    PROC rMoveWeld()
        IF nMode=1 THEN
            stCommand:="Weld1";
            WaitUntil stReact=["WeldOk","WeldOk","WeldOk"]OR stReact=["Error_Arc_Touch","Error_Arc_Touch","Error_Arc_Touch"];
            IF stReact=["Error_Arc_Touch","Error_Arc_Touch","Error_Arc_Touch"]rMoveHome_Head;

            stCommand:="";
            WaitUntil stReact=["Ready","Ready","Ready"];
        ELSEIF nMode=2 THEN
            stCommand:="Weld2";
            WaitUntil stReact=["WeldOk","WeldOk","WeldOk"]OR stReact=["Error_Arc_Touch","Error_Arc_Touch","Error_Arc_Touch"];
            IF stReact=["Error_Arc_Touch","Error_Arc_Touch","Error_Arc_Touch"]rMoveHome_Head;

            stCommand:="";
            WaitUntil stReact=["Ready","Ready","Ready"];
        ELSE
            stCommand:="Weld";
            WaitUntil stReact=["WeldOk","WeldOk","WeldOk"]OR stReact=["Error_Arc_Touch","Error_Arc_Touch","Error_Arc_Touch"];
            IF stReact=["Error_Arc_Touch","Error_Arc_Touch","Error_Arc_Touch"]rMoveHome_Head;

            stCommand:="";
            WaitUntil stReact=["Ready","Ready","Ready"];

        ENDIF
    ENDPROC

    PROC rNozzleClean(string Mode)
        VAR jointgroup jgCurrent;
        rGantry_C_Home;
        bNozzleCleanCut:=TRUE;
        rMeasurementHomeCheck;
        TEST Mode
        CASE "R1":
            rWirecutMove 1;
        CASE "R2":
            rWirecutMove 2;
        CASE "R1&R2":
            rWirecutMove 3;
        DEFAULT:
        ENDTEST
        bNozzleCleanCut:=FALSE;
        TEST Mode
        CASE "R1":
            rNozzleClean_R1;
        CASE "R2":
            rNozzleClean_R2;
        CASE "R1&R2":
            jgCurrent:=MergeJgWith();
            IF jgCurrent.JointG.extax.eax_d<0 THEN
                rNozzleClean_R1;
                rNozzleClean_R2;
            ELSE
                rNozzleClean_R2;
                rNozzleClean_R1;
            ENDIF
        DEFAULT:
        ENDTEST

    ENDPROC

    PROC rNozzleClean_R1()
        VAR jointgroup jgTemp;
        VAR speeddata vTemp:=[25,25,400,25];
        jgTemp:=MergeJgWith();
        jgTemp.JointG.extax.eax_b:=jNozzleClean_R1.extax.eax_b;
        jgTemp.JointG.extax.eax_c:=jNozzleClean_R1.extax.eax_c;
        jgTemp.JointG.extax.eax_d:=jNozzleClean_R1.extax.eax_d;
        MoveJgJ MergeJgWith(\Gantry:=jgTemp.JointG),vTemp,fine;
        WaitRob\InPos;
        nR_Angle:=jgTemp.JointG.extax.eax_d;
        stCommand:="NozzleClean_R1";
        WaitUntil stReact=["NozzleClean_R1_Ok","Ready","Ready"];
        stCommand:="";
        WaitUntil stReact=["Ready","Ready","Ready"];
    ENDPROC

    PROC rNozzleClean_R2()
        VAR jointgroup jgTemp;
        VAR speeddata vTemp:=[25,25,400,25];
        jgTemp:=MergeJgWith();
        jgTemp.JointG.extax.eax_b:=jNozzleClean_R2.extax.eax_b;
        jgTemp.JointG.extax.eax_c:=jNozzleClean_R2.extax.eax_c;
        jgTemp.JointG.extax.eax_d:=jNozzleClean_R2.extax.eax_d;
        MoveJgJ MergeJgWith(\Gantry:=jgTemp.JointG),vTemp,fine;
        WaitRob\InPos;
        nR_Angle:=jgTemp.JointG.extax.eax_d;
        stCommand:="NozzleClean_R2";
        WaitUntil stReact=["Ready","NozzleClean_R2_Ok","Ready"];
        stCommand:="";
        WaitUntil stReact=["Ready","Ready","Ready"];
    ENDPROC

    PROC rTpRoutine()
        VAR num n;
        VAR num nn;
        VAR num nGantryX;
        VAR num nGantryY;
        VAR num nGantryZ;
        VAR num nRobotAxis1;
        VAR num nRobotAxis2;
        VAR num nRobotAxis3;
        VAR num nRobotAxis4;
        VAR num nRobotAxis5;
        VAR num nRobotAxis6;
        VAR jointtarget rEmptyJoint;

        gStart:
        TPErase;
        TPReadFK n,"Did you want TP Manual Mode or Auto Mode?","Manual",stEmpty,stEmpty,stEmpty,"Auto";

        IF n=5 GOTO gAuto;
        TPReadFK n,"What Position?","Manual Pos",stEmpty,"Repair Pos","Home Pos","Menu";

        TEST n
        CASE 1:
            gMoving:
            TPReadFK n,"What do you want?","Gantry Move",stEmpty,stEmpty,"Robot Move","Menu";

            IF n=1 THEN
                TPReadNum nGantryX,"Gantry X";
                TPReadNum nGantryY,"Gantry Y";
                TPReadNum nGantryZ,"Gantry Z";
                TPErase;
                TPWrite "X"+ValToStr(nGantryX)+"Y"+ValToStr(nGantryY)+"Z"+ValToStr(nGantryZ);
                TPReadFK n,"Right?","Yes",stEmpty,stEmpty,"No","Menu";

                IF n=1 THEN
                    rEmptyJoint:=CJointT();
                    rEmptyJoint.extax.eax_a:=nHomeGantryX+nGantryX;
                    rEmptyJoint.extax.eax_b:=nHomeGantryX+nGantryX;
                    rEmptyJoint.extax.eax_c:=nHomeGantryY-nGantryY;
                    rEmptyJoint.extax.eax_d:=nHomeGantryZ-nGantryZ;

                    TPErase;
                    TPWrite "!!!!!!!!!!!!!!!!!!!!!!!!!";
                    TPWrite "BE Carful! Gantry Moving!";
                    TPWrite "!!!!!!!!!!!!!!!!!!!!!!!!!";
                    WaitTime 0.3;
                    MoveAbsJ rEmptyJoint,v300,fine,tool0;

                    TPErase;
                    TPWrite "!!!!!!!!!!!!!!!!!!!!!!!!!";
                    TPWrite "!!!! Gantry Arrived !!!!!";
                    TPWrite "!!!!!!!!!!!!!!!!!!!!!!!!!";
                    WaitTime 0.3;

                    GOTO gMoving;

                ELSEIF n=4 THEN
                    TPErase;
                    TPWrite "Go To Select";
                    WaitTime 0.3;
                    GOTO gMoving;
                ELSE
                    TPErase;
                    TPWrite "Go To Menu";
                    WaitTime 0.3;
                    GOTO gStart;
                ENDIF

            ELSEIF n=4 THEN
                TPErase;
                TPReadNum nRobotAxis1,"Robot Axis 1";
                TPReadNum nRobotAxis2,"Robot Axis 2";
                TPReadNum nRobotAxis3,"Robot Axis 3";
                TPReadNum nRobotAxis4,"Robot Axis 4";
                TPReadNum nRobotAxis5,"Robot Axis 5";
                TPReadNum nRobotAxis6,"Robot Axis 6";

                TPErase;
                TPWrite "Axis 1 : "+ValToStr(nRobotAxis1)+"Axis 2 : "+ValToStr(nRobotAxis2)+"Axis 3 : "+ValToStr(nRobotAxis3);
                TPWrite "Axis 4 : "+ValToStr(nRobotAxis4)+"Axis 5 : "+ValToStr(nRobotAxis5)+"Axis 6 : "+ValToStr(nRobotAxis6);
                TPReadFK n,"Right?","Yes",stEmpty,stEmpty,"No","Menu";

                IF n=1 THEN
                    rEmptyJoint:=CJointT();
                    rEmptyJoint.robax.rax_1:=nRobotAxis1;
                    rEmptyJoint.robax.rax_2:=nRobotAxis2;
                    rEmptyJoint.robax.rax_3:=nRobotAxis3;
                    rEmptyJoint.robax.rax_4:=nRobotAxis4;
                    rEmptyJoint.robax.rax_5:=nRobotAxis5;
                    rEmptyJoint.robax.rax_6:=nRobotAxis6;

                    TPErase;
                    TPWrite "!!!!!!!!!!!!!!!!!!!!!!!!!";
                    TPWrite "BE Carful! Robot  Moving!";
                    TPWrite "!!!!!!!!!!!!!!!!!!!!!!!!!";
                    WaitTime 0.3;
                    MoveAbsJ rEmptyJoint,v300,fine,tool0;

                    TPErase;
                    TPWrite "!!!!!!!!!!!!!!!!!!!!!!!!!";
                    TPWrite "!!!! Robot  Arrived !!!!!";
                    TPWrite "!!!!!!!!!!!!!!!!!!!!!!!!!";
                    WaitTime 0.3;

                    GOTO gMoving;

                ELSEIF n=4 THEN
                    TPErase;
                    TPWrite "Go To Select";
                    WaitTime 0.3;
                    GOTO gMoving;
                ELSE
                    TPErase;
                    TPWrite "Go To Menu";
                    WaitTime 0.3;
                    GOTO gStart;
                ENDIF

            ELSE
                TPErase;
                TPWrite "Go To Menu";
                WaitTime 0.3;
                GOTO gStart;
            ENDIF


        CASE 3:

            gRepairStart:
            TPErase;
            TPReadFK n,"What do you want to do?","Change Repair Pos",stEmpty,stEmpty,"Move Repair","Menu";


            IF n=1 THEN
                TPReadFK n,"Did you Change Here?","Yes",stEmpty,stEmpty,"NO","Menu";
                IF n=5 GOTO gStart;
                WaitRob\ZeroSpeed;
                ClearPath;
                rEmptyJoint:=CJointT();
                TPErase;
                TPWrite "Gantry Check";
                TPWrite "Gantry X : "+ValToStr(rEmptyJoint.extax.eax_a);
                TPWrite "Gantry Y : "+ValToStr(nHomeGantryY-rEmptyJoint.extax.eax_c);
                TPWrite "Gantry Z : "+ValToStr(nHomeGantryZ-rEmptyJoint.extax.eax_d);
                WaitTime 0.3;

                TPReadFK n,"Right?","Yes",stEmpty,stEmpty,stEmpty,"No";
                IF n=5 GOTO gRepairStart;

                TPErase;
                TPWrite "Robot Axis 1 : "+ValToStr(rEmptyJoint.robax.rax_1)+"Robot Axis 2 : "+ValToStr(rEmptyJoint.robax.rax_2);
                TPWrite "Robot Axis 3 : "+ValToStr(rEmptyJoint.robax.rax_3)+"Robot Axis 4 : "+ValToStr(rEmptyJoint.robax.rax_4);
                TPWrite "Robot Axis 5 : "+ValToStr(rEmptyJoint.robax.rax_5)+"Robot Axis 6 : "+ValToStr(rEmptyJoint.robax.rax_6);

                TPReadFK n,"Right?","Yes",stEmpty,stEmpty,stEmpty,"No";

                IF n=5 GOTO gRepairStart;
                IF n=1 THEN
                    TPReadFK n,"Did you want Save Repair Position?","Yes",stEmpty,stEmpty,stEmpty,"No";
                    IF n=5 GOTO gRepairStart;
                    TPErase;
                    TPWrite "Save Repair Position";
                    jRepairJoint:=rEmptyJoint;
                    WaitTime 0.3;
                    GOTO gRepairStart;
                ENDIF

            ELSEIF n=4 THEN
                MoveAbsJ jRepairJoint,v300,fine,tool0;

            ELSE
                TPErase;
                TPWrite "Go To Manu";
                WaitTime 0.3;
                GOTO gStart;

            ENDIF

        CASE 4:

            gHomeStart:
            TPReadFK n,"What do you want?","Change Home Pos",stEmpty,stEmpty,"Move Home","Menu";

            IF n=1 THEN

                TPReadFK n,"Did you Change Here?","Yes",stEmpty,stEmpty,"NO","Menu";
                IF n=5 GOTO gStart;
                WaitRob\ZeroSpeed;
                ClearPath;
                rEmptyJoint:=CJointT();
                TPErase;
                TPWrite "Gantry Check";
                TPWrite "Gantry X : "+ValToStr(rEmptyJoint.extax.eax_a);
                TPWrite "Gantry Y : "+ValToStr(nHomeGantryY-rEmptyJoint.extax.eax_c);
                TPWrite "Gantry Z : "+ValToStr(nHomeGantryZ-rEmptyJoint.extax.eax_d);
                WaitTime 0.3;

                TPReadFK n,"Right?","Yes",stEmpty,stEmpty,stEmpty,"No";
                IF n=5 GOTO gHomeStart;

                TPErase;
                TPWrite "Robot Axis 1 : "+ValToStr(rEmptyJoint.robax.rax_1)+"Robot Axis 2 : "+ValToStr(rEmptyJoint.robax.rax_2);
                TPWrite "Robot Axis 3 : "+ValToStr(rEmptyJoint.robax.rax_3)+"Robot Axis 4 : "+ValToStr(rEmptyJoint.robax.rax_4);
                TPWrite "Robot Axis 5 : "+ValToStr(rEmptyJoint.robax.rax_5)+"Robot Axis 6 : "+ValToStr(rEmptyJoint.robax.rax_6);

                TPReadFK n,"Right?","Yes",stEmpty,stEmpty,stEmpty,"No";
                IF n=5 GOTO gHomeStart;
                IF n=1 THEN
                    TPReadFK n,"Did you want Save Home Position?","Yes",stEmpty,stEmpty,stEmpty,"No";
                    IF n=5 GOTO gHomeStart;
                    TPErase;
                    TPWrite "Save Home Position";
                    jHomeJoint:=rEmptyJoint;
                    WaitTime 0.3;
                ENDIF
                GOTO gHomeStart;

            ELSEIF n=4 THEN
                TPWrite "Go Home Position";
                rMoveHome;
                TPWrite "Arrived Homoe Position Go to Menu";
            ELSE

                TPWrite "Go To Menu";
                WaitTime 0.3;
                GOTO gStart;

            ENDIF

        CASE 5:
            TPWrite "Go To Menu";
            WaitTime 0.3;
            GOTO gStart;
        ENDTEST

        gAuto:

    ENDPROC

    PROC rWirecut(num nRbt_No)
        bWirecut:=[FALSE,FALSE,FALSE];
        IF (sdo_Rob_1_JgHome=1 AND sdo_Rob_2_JgHome=1) OR (sdo_Rob_1_MoveHome=1 AND sdo_Rob_2_MoveHome=1) OR (sdo_Rob_1_WirecutHome=1 AND sdo_Rob_2_WirecutHome=1) THEN
        ELSE
            rMeasurementHomeCheck;
        ENDIF
        IF sdo_Rob_1_JgHome=1 AND sdo_Rob_2_JgHome=1 THEN
            bWirecut:=[TRUE,FALSE,FALSE];
            IF nRbt_No=0 OR nRbt_No=1 THEN
                Wirecut\R1;
                WaitUntil stReact{1}="WireCutOk";
                stCommand:="";
                WaitUntil stReact{1}="Ready";
            ENDIF
            IF nRbt_No=0 OR nRbt_No=2 THEN
                WireCut\R2;
                WaitUntil stReact{2}="WireCutOk";
                stCommand:="";
                WaitUntil stReact{2}="Ready";
            ENDIF
            IF nRbt_No=3 THEN
                bWireCutSync:=TRUE;
                stCommand:="WireCutR1_R2";
                WaitUntil stReact{1}="WireCutOk" AND stReact{2}="WireCutOk";
                stCommand:="";
                WaitUntil stReact{1}="Ready" AND stReact{2}="Ready";
                bWireCutSync:=FALSE;
            ENDIF
        ENDIF
        IF sdo_Rob_1_MoveHome=1 AND sdo_Rob_2_MoveHome=1 THEN
            bWirecut:=[FALSE,TRUE,FALSE];
            IF nRbt_No=0 OR nRbt_No=1 THEN
                WirecutMove\R1;
                WaitUntil stReact{1}="WireCutOk";
                stCommand:="";
                WaitUntil stReact{1}="Ready";
            ENDIF
            IF nRbt_No=0 OR nRbt_No=2 THEN
                WireCutMove\R2;
                WaitUntil stReact{2}="WireCutOk";
                stCommand:="";
                WaitUntil stReact{2}="Ready";
            ENDIF
            IF nRbt_No=3 THEN
                bWireCutSync:=TRUE;
                stCommand:="WireCutMoveR1_R2";
                WaitUntil stReact{1}="WireCutOk" AND stReact{2}="WireCutOk";
                stCommand:="";
                WaitUntil stReact{1}="Ready" AND stReact{2}="Ready";
                bWireCutSync:=FALSE;
            ENDIF
        ENDIF
        IF sdo_Rob_1_WirecutHome=1 AND sdo_Rob_2_WirecutHome=1 THEN
            bWirecut:=[FALSE,FALSE,TRUE];
            IF nRbt_No=0 OR nRbt_No=1 THEN
                WirecutShot\R1;
                WaitUntil stReact{1}="WireCutOk";
                stCommand:="";
                WaitUntil stReact{1}="Ready";
            ENDIF
            IF nRbt_No=0 OR nRbt_No=2 THEN
                WireCutShot\R2;
                WaitUntil stReact{2}="WireCutOk";
                stCommand:="";
                WaitUntil stReact{2}="Ready";
            ENDIF
            IF nRbt_No=3 THEN
                bWireCutSync:=TRUE;
                stCommand:="WireCutShotR1_R2";
                WaitUntil stReact{1}="WireCutOk" AND stReact{2}="WireCutOk";
                stCommand:="";
                WaitUntil stReact{1}="Ready" AND stReact{2}="Ready";
                bWireCutSync:=FALSE;
            ENDIF
        ENDIF
        WaitUntil stReact=["Ready","Ready","Ready"];

    ENDPROC

    PROC rWirecutShot(num nRbt_No)

        IF nRbt_No=0 OR nRbt_No=1 THEN
            WirecutShot\R1;
            WaitUntil stReact{1}="WireCutOk";
            stCommand:="";
            WaitUntil stReact{1}="Ready";
        ENDIF
        IF nRbt_No=0 OR nRbt_No=2 THEN
            WireCutShot\R2;
            WaitUntil stReact{2}="WireCutOk";
            stCommand:="";
            WaitUntil stReact{2}="Ready";
        ENDIF
        IF nRbt_No=3 THEN
            bWireCutSync:=TRUE;
            stCommand:="WireCutShotR1_R2";
            WaitUntil stReact{1}="WireCutOk" AND stReact{2}="WireCutOk";
            stCommand:="";
            WaitUntil stReact{1}="Ready" AND stReact{2}="Ready";
            bWireCutSync:=FALSE;
        ENDIF

        WaitUntil stReact=["Ready","Ready","Ready"];

    ENDPROC

    PROC rWirecutMove(num nRbt_No)

        IF nRbt_No=0 OR nRbt_No=1 THEN
            WirecutMove\R1;
            WaitUntil stReact{1}="WireCutOk";
            stCommand:="";
            WaitUntil stReact{1}="Ready";
        ENDIF
        IF nRbt_No=0 OR nRbt_No=2 THEN
            WireCutMove\R2;
            WaitUntil stReact{2}="WireCutOk";
            stCommand:="";
            WaitUntil stReact{2}="Ready";
        ENDIF
        IF nRbt_No=3 THEN
            bWireCutSync:=TRUE;
            stCommand:="WireCutMoveR1_R2";
            WaitUntil stReact{1}="WireCutOk" AND stReact{2}="WireCutOk";
            stCommand:="";
            WaitUntil stReact{1}="Ready" AND stReact{2}="Ready";
            bWireCutSync:=FALSE;
        ENDIF

        WaitUntil stReact=["Ready","Ready","Ready"];

    ENDPROC

    PROC rEdgeDataCheck()
        IF edgeStart{1}.Breadth<=0 edgeStart{1}.Breadth:=50;
        IF edgeStart{1}.Height<=0 edgeStart{1}.Height:=50;
        IF edgeStart{2}.Breadth<=0 edgeStart{2}.Breadth:=50;
        IF edgeStart{2}.Height<=0 edgeStart{2}.Height:=50;
        IF edgeEnd{1}.Breadth<=0 edgeEnd{1}.Breadth:=50;
        IF edgeEnd{1}.Height<=0 edgeEnd{1}.Height:=50;
        IF edgeEnd{2}.Breadth<=0 edgeEnd{2}.Breadth:=50;
        IF edgeEnd{2}.Height<=0 edgeEnd{2}.Height:=50;
    ENDPROC

    PROC rMoveHome_Head()

        WaitUntil stReact=["Error_Arc_Touch","Error_Arc_Touch","Error_Arc_Touch"];
        stCommand:="Error_Arc_Touch";
        WaitUntil stReact=["","",""];
        stCommand:="";
        WaitUntil stReact=["","",""];
        nErrorCmd:=1;
        ExitCycle;

    ENDPROC

    PROC rWireReplacementMode()
        VAR jointgroup jTempReadyGroup;
        VAR num nTempChangPos;
        VAR num nMaxHeight;
        !!!!!!==MoveToHome==,[
        rMeasurementHomeCheck;

        jTempReadyGroup:=MergeJgWith();
        jTempReadyGroup.JointG.extax.eax_b:=Limit(0,5300,nLimitY_Positive-nMaintenanceYPos);
        jTempReadyGroup.JointG.extax.eax_d:=0;
        MoveJgJ MergeJgWith(\Gantry:=jTempReadyGroup.JointG),vTargetSpeed,z200;

        jTempReadyGroup.JointG.extax.eax_c:=700;
        MoveJgJ MergeJgWith(\Gantry:=jTempReadyGroup.JointG),vTargetSpeed,z200;

        RETURN ;
    ENDPROC

    PROC rArcErrorGantryDown()
        VAR jointgroup jTempReadyGroup;
        VAR num nTempGantryHeight;
        VAR num nTempPartHeightTemp;
        jTempReadyGroup:=MergeJgWith();
        nTempPartHeightTemp:=max(max(nMaxPartHeightNearArray{1},nMaxPartHeightNearArray{2}),nMaxPartHeightNearArray{3});

        nTempGantryHeight:=nHomeGantryZ-(900+nTempPartHeightTemp);
        jTempReadyGroup.JointG.extax.eax_c:=nTempGantryHeight;
        jTempReadyGroup.JointG.extax.eax_c:=Limit(0,1000,jTempReadyGroup.JointG.extax.eax_c);
        MoveJgJ MergeJgWith(\Gantry:=jTempReadyGroup.JointG),vTargetSpeed,z200;
    ENDPROC

    PROC rMeasurementHomeCheck()
        VAR jointgroup jMeasurementHomeGroup;
        VAR bool bHomeCheck:=FALSE;
        bHomeCheck:=FALSE;
        jMeasurementHomeGroup:=MergeJgWith();
        IF abs(jMeasurementHomeGroup.Joint1.robax.rax_1-jgMeasurementHome.Joint1.robax.rax_1)>1 bHomeCheck:=TRUE;
        IF abs(jMeasurementHomeGroup.Joint1.robax.rax_2-jgMeasurementHome.Joint1.robax.rax_2)>1 bHomeCheck:=TRUE;
        IF abs(jMeasurementHomeGroup.Joint1.robax.rax_3-jgMeasurementHome.Joint1.robax.rax_3)>1 bHomeCheck:=TRUE;
        IF abs(jMeasurementHomeGroup.Joint1.robax.rax_4-jgMeasurementHome.Joint1.robax.rax_4)>1 bHomeCheck:=TRUE;
        IF abs(jMeasurementHomeGroup.Joint1.robax.rax_5-jgMeasurementHome.Joint1.robax.rax_5)>1 bHomeCheck:=TRUE;
        IF abs(jMeasurementHomeGroup.Joint1.robax.rax_6-jgMeasurementHome.Joint1.robax.rax_6)>1 bHomeCheck:=TRUE;
        IF abs(jMeasurementHomeGroup.Joint2.robax.rax_1-jgMeasurementHome.Joint2.robax.rax_1)>1 bHomeCheck:=TRUE;
        IF abs(jMeasurementHomeGroup.Joint2.robax.rax_2-jgMeasurementHome.Joint2.robax.rax_2)>1 bHomeCheck:=TRUE;
        IF abs(jMeasurementHomeGroup.Joint2.robax.rax_3-jgMeasurementHome.Joint2.robax.rax_3)>1 bHomeCheck:=TRUE;
        IF abs(jMeasurementHomeGroup.Joint2.robax.rax_4-jgMeasurementHome.Joint2.robax.rax_4)>1 bHomeCheck:=TRUE;
        IF abs(jMeasurementHomeGroup.Joint2.robax.rax_5-jgMeasurementHome.Joint2.robax.rax_5)>1 bHomeCheck:=TRUE;
        IF abs(jMeasurementHomeGroup.Joint2.robax.rax_6-jgMeasurementHome.Joint2.robax.rax_6)>1 bHomeCheck:=TRUE;

        IF bHomeCheck=TRUE THEN
            rByTaskMoveToRobotHome 1;
        ELSE
            jMeasurementHomeGroup.JointG.extax.eax_c:=0;
            MoveJgJ jMeasurementHomeGroup,vTargetSpeed,fine;
        ENDIF
    ENDPROC

    PROC rjgWireCutHomeCheck()
        VAR jointgroup jWirecutHomeGroup;
        VAR bool bHomeCheck:=FALSE;
        bHomeCheck:=FALSE;
        jWirecutHomeGroup:=MergeJgWith();

        IF abs(jWirecutHomeGroup.Joint1.robax.rax_1-jgWireCutHome.Joint1.robax.rax_1)>1 bHomeCheck:=TRUE;
        IF abs(jWirecutHomeGroup.Joint1.robax.rax_2-jgWireCutHome.Joint1.robax.rax_2)>1 bHomeCheck:=TRUE;
        IF abs(jWirecutHomeGroup.Joint1.robax.rax_3-jgWireCutHome.Joint1.robax.rax_3)>1 bHomeCheck:=TRUE;
        IF abs(jWirecutHomeGroup.Joint1.robax.rax_4-jgWireCutHome.Joint1.robax.rax_4)>1 bHomeCheck:=TRUE;
        IF abs(jWirecutHomeGroup.Joint1.robax.rax_5-jgWireCutHome.Joint1.robax.rax_5)>1 bHomeCheck:=TRUE;
        IF abs(jWirecutHomeGroup.Joint1.robax.rax_6-jgWireCutHome.Joint1.robax.rax_6)>1 bHomeCheck:=TRUE;
        IF abs(jWirecutHomeGroup.Joint2.robax.rax_1-jgWireCutHome.Joint2.robax.rax_1)>1 bHomeCheck:=TRUE;
        IF abs(jWirecutHomeGroup.Joint2.robax.rax_2-jgWireCutHome.Joint2.robax.rax_2)>1 bHomeCheck:=TRUE;
        IF abs(jWirecutHomeGroup.Joint2.robax.rax_3-jgWireCutHome.Joint2.robax.rax_3)>1 bHomeCheck:=TRUE;
        IF abs(jWirecutHomeGroup.Joint2.robax.rax_4-jgWireCutHome.Joint2.robax.rax_4)>1 bHomeCheck:=TRUE;
        IF abs(jWirecutHomeGroup.Joint2.robax.rax_5-jgWireCutHome.Joint2.robax.rax_5)>1 bHomeCheck:=TRUE;
        IF abs(jWirecutHomeGroup.Joint2.robax.rax_6-jgWireCutHome.Joint2.robax.rax_6)>1 bHomeCheck:=TRUE;

        IF bHomeCheck=TRUE THEN
            rByTaskMoveToRobotHome 2;
        ELSE
            jWirecutHomeGroup.JointG.extax.eax_c:=0;
            MoveJgJ jWirecutHomeGroup,vTargetSpeed,fine;
        ENDIF
    ENDPROC

    PROC rByTaskMoveToRobotHome(num nHomeNo)
        VAR jointgroup jgEmptyTarget;
        VAR jointtarget jTempG;
        VAR num ntemp;

        stCommand:="checkpos";
        waituntil stReact=["checkposok","checkposok","checkposok"];
        stCommand:="";
        waituntil stReact=["Ready","Ready","Ready"];

        jgEmptyTarget.Joint1:=CJointT(\TaskName:="T_Rob1");
        jgEmptyTarget.Joint2:=CJointT(\TaskName:="T_Rob2");
        jgEmptyTarget.JointG:=CJointT(\TaskName:="T_Gantry");
        jgEmptyTarget.JointG.extax.eax_c:=0;
        MoveJgJ jgEmptyTarget,vTargetSpeed,fine;

        jgEmptyTarget.Joint1.robax.rax_2:=-90;
        jgEmptyTarget.Joint1.robax.rax_3:=55;
        jgEmptyTarget.Joint2.robax.rax_2:=-90;
        jgEmptyTarget.Joint2.robax.rax_3:=55;
        MoveJgJ jgEmptyTarget,vTargetSpeed,fine;

        jgEmptyTarget.Joint1.robax.rax_5:=0;
        jgEmptyTarget.Joint2.robax.rax_5:=0;
        MoveJgJ jgEmptyTarget,vTargetSpeed,fine;
        IF nHomeNo=1 THEN
            jgEmptyTarget.Joint1.robax.rax_1:=jgMeasurementHome.Joint1.robax.rax_1;
            jgEmptyTarget.Joint2.robax.rax_1:=jgMeasurementHome.Joint2.robax.rax_1;
        ELSEIF nHomeNo=2 THEN
            jgEmptyTarget.Joint1.robax.rax_1:=jgWireCutHome.Joint1.robax.rax_1;
            jgEmptyTarget.Joint2.robax.rax_1:=jgWireCutHome.Joint2.robax.rax_1;
        ENDIF
        IF bNozzleCleanCut=FALSE jgEmptyTarget.JointG.extax.eax_d:=0;
        MoveJgJ jgEmptyTarget,vTargetSpeed,fine;

        jgEmptyTarget.Joint1:=CJointT(\TaskName:="T_Rob1");
        jgEmptyTarget.Joint2:=CJointT(\TaskName:="T_Rob2");
        jgEmptyTarget.JointG:=CJointT(\TaskName:="T_Gantry");
        IF nHomeNo=1 THEN
            jgEmptyTarget.Joint1.robax:=jgMeasurementHome.Joint1.robax;
            jgEmptyTarget.Joint2.robax:=jgMeasurementHome.Joint2.robax;
        ELSEIF nHomeNo=2 THEN
            jgEmptyTarget.Joint1.robax:=jgWireCutHome.Joint1.robax;
            jgEmptyTarget.Joint2.robax:=jgWireCutHome.Joint2.robax;
        ENDIF
        MoveJgJ jgEmptyTarget,vTargetSpeed,fine;

        RETURN ;
    ENDPROC

    PROC rWarm_Up()

        VAR speeddata vWarmUp_Speed;
        VAR num i:=0;
        VAR num nWarmUp_Distance_X;
        VAR num nWarmUp_Distance_Y;
        VAR num nWarmUp_Distance_Z;
        VAR num nWarmUp_Distance_R;
        VAR num nTempDistance:=0;
        VAR clock clWarmUp;
        VAR bool bWarmUpComplete:=FALSE;
        VAR jointgroup jgWarmUpTargetpos;



        !..... Userset Gantry_X .........
        !        nWarmUp_Target_X:=-9000;
        !................................
        jgWarmUpTargetpos:=jgHomeJoint;
        jgWarmUpTargetpos.JointG.extax.eax_a:=nWarmUp_Target_X;
        jgWarmUpTargetpos.JointG.extax.eax_f:=nWarmUp_Target_X;

        jgTarget:=MergeJgWith();
        jgTarget.JointG:=jgWarmUpTargetpos.JointG;
        jgTarget.JointG.extax.eax_d:=90;

        vWarmUp_Speed:=[300,300,10,10];
        ClkReset clWarmUp;
        ClkStart clWarmUp;

        WHILE bWarmUpComplete=FALSE DO

            jgWarm_Up:=MergeJgWith();

            ! eax_a
            IF jgWarm_Up.JointG.extax.eax_a<jgWarmUpTargetpos.JointG.extax.eax_a+149 AND jgWarm_Up.JointG.extax.eax_a>jgWarmUpTargetpos.JointG.extax.eax_a-149 THEN
                jgTarget.JointG.extax.eax_a:=jgWarmUpTargetpos.JointG.extax.eax_a-150;
            ELSE
                IF jgWarm_Up.JointG.extax.eax_a<jgWarmUpTargetpos.JointG.extax.eax_a-150 jgTarget.JointG.extax.eax_a:=jgWarmUpTargetpos.JointG.extax.eax_a+150;
            ENDIF
            nWarmUp_Distance_X:=jgTarget.JointG.extax.eax_a-jgWarm_Up.JointG.extax.eax_a;
            IF nWarmUp_Distance_X>0 THEN
                nTempDistance:=100;
            ELSE
                nTempDistance:=-100;
            ENDIF
            jgWarm_Up.JointG.extax.eax_a:=jgWarm_Up.JointG.extax.eax_a+nTempDistance;
            jgWarm_Up.JointG.extax.eax_f:=jgWarm_Up.JointG.extax.eax_f+nTempDistance;

            ! eax_b
            IF jgWarm_Up.JointG.extax.eax_b>149 jgTarget.JointG.extax.eax_b:=0;
            IF jgWarm_Up.JointG.extax.eax_b<1 jgTarget.JointG.extax.eax_b:=150;
            nWarmUp_Distance_Y:=jgTarget.JointG.extax.eax_b-jgWarm_Up.JointG.extax.eax_b;
            IF nWarmUp_Distance_Y>0 THEN
                nTempDistance:=100;
            ELSE
                nTempDistance:=-100;
            ENDIF
            jgWarm_Up.JointG.extax.eax_b:=jgWarm_Up.JointG.extax.eax_b+nTempDistance;

            ! eax_c
            IF jgWarm_Up.JointG.extax.eax_c<1 jgTarget.JointG.extax.eax_c:=100;
            IF jgWarm_Up.JointG.extax.eax_c>99 jgTarget.JointG.extax.eax_c:=0;
            nWarmUp_Distance_Z:=jgTarget.JointG.extax.eax_c-jgWarm_Up.JointG.extax.eax_c;
            IF nWarmUp_Distance_Z>0 THEN
                nTempDistance:=100;
            ELSE
                nTempDistance:=-100;
            ENDIF
            jgWarm_Up.JointG.extax.eax_c:=jgWarm_Up.JointG.extax.eax_c+nTempDistance;

            ! eax_d
            IF jgWarm_Up.JointG.extax.eax_d<-81 jgTarget.JointG.extax.eax_d:=90;
            IF jgWarm_Up.JointG.extax.eax_d>81 jgTarget.JointG.extax.eax_d:=-90;
            nWarmUp_Distance_R:=jgTarget.JointG.extax.eax_d-jgWarm_Up.JointG.extax.eax_d;
            IF nWarmUp_Distance_R>0 THEN
                nTempDistance:=10;
            ELSE
                nTempDistance:=-10;
            ENDIF
            jgWarm_Up.JointG.extax.eax_d:=jgWarm_Up.JointG.extax.eax_d+nTempDistance;

            !  move
            jgWarm_Up.JointG.extax.eax_b:=Limit(0,5300,jgWarm_Up.JointG.extax.eax_b);
            jgWarm_Up.JointG.extax.eax_c:=Limit(0,100,jgWarm_Up.JointG.extax.eax_c);
            jgWarm_Up.JointG.extax.eax_d:=Limit(-90,90,jgWarm_Up.JointG.extax.eax_d);
            MoveJgJ MergeJgWith(\Gantry:=jgWarm_Up.JointG),vWarmUp_Speed,fine;
            vWarmUp_Speed.v_reax:=vWarmUp_Speed.v_reax+0.1;
            vWarmUp_Speed.v_leax:=vWarmUp_Speed.v_leax+0.5;
            IF vWarmUp_Speed.v_reax>25 vWarmUp_Speed.v_reax:=25;
            IF vWarmUp_Speed.v_leax>250 vWarmUp_Speed.v_leax:=250;
            nWarmUpTime:=ClkRead(clWarmUp);
            IF nWarmUpTime>nWarmUpCycle bWarmUpComplete:=TRUE;
        ENDWHILE
        ClkStop clWarmUp;
        RETURN ;
    ENDPROC

    PROC rGantry_C_Home()
        VAR jointgroup jgGantry_C_Home;
        jgGantry_C_Home:=MergeJgWith();
        jgGantry_C_Home.JointG.extax.eax_c:=0;
        MoveJgJ MergeJgWith(\Gantry:=jgGantry_C_Home.JointG),vTargetSpeed,fine;
        WaitRob\InPos;
        WaitRob\ZeroSpeed;
    ENDPROC

    PROC rLdsCheck()

        rGantry_C_Home;
        rMeasurementHomeCheck;

        stCommand:="LdsCheck";
        WaitUntil(stReact=["Ready","Ready","LdsCheck_Ok"]);

        stCommand:="";
        WaitUntil stReact=["Ready","Ready","Ready"];

        IF bLDS_Origin=FALSE and (abs(nDiffGantryX)>1 OR abs(nDiffGantryY)>1 OR abs(nDiffGantryZ)>1) THEN
            ErrLog 4811,"LDS_OutRangeError","","","","";
            !          WaitUntil pi19_=1 OR pi20_=1;
            !          IF pi19_=1 GOTO LabalReturn;
            !          IF pi20_=1 rSettingInitialize;
        ELSE
            rSettingInitialize;
        ENDIF

    ENDPROC

    PROC rTcp_Inspect()
        VAR jointtarget jMoveGantry;
        VAR jointgroup jTempReadyGroup;
        VAR jointtarget jWeldPrepareR1{10};
        VAR jointtarget jWeldPrepareR2{10};
        VAR jointtarget jTempGantry{2};
        VAR num nGantryAngel;
        VAR robtarget pDefineWeldPos;
        VAR jointgroup jTempGroup;

        posStart.x:=tOrder.Tcp_X;
        posStart.y:=tOrder.Tcp_Y;
        posStart.z:=tOrder.Tcp_Z;
        nGantryAngel:=tOrder.Tcp_Angle;
        posEnd:=posStart;
        posEnd.x:=posEnd.x+100;
        nStartThick:=0;
        nEndThick:=0;
        posStartLast:=posStart;
        posEndLast:=posEnd;
        nLengthWeldLine:=0;
        !!!!!!

        rDefineWobjWeldLineTcp posStart,posEnd;
        nBreakPoint:=[0,0];
        !        rDefineWeldPosR1;
        pDefineWeldPos:=pNull;
        pDefineWeldPos.trans:=[0,0,0];
        pDefineWeldPos.robconf:=[0,0,0,1];
        pDefineWeldPos.rot:=[0.5,0.5,-0.5,0.5];
        pDefineWeldPos:=RelTool(pDefineWeldPos,0,0,0\Rx:=0\Ry:=-45);
        Welds1{1}.position:=pDefineWeldPos;
        pDefineWeldPos.rot:=[0.5,-0.5,-0.5,-0.5];
        pDefineWeldPos:=RelTool(pDefineWeldPos,0,0,0\Rx:=0\Ry:=-45);
        Welds2{1}.position:=pDefineWeldPos;
        WeldsG{1}.position.trans:=CalcPosOnLine(posStart,posEnd,0);
        WeldsG{1}.position.trans.z:=WeldsG{1}.position.trans.z+nRobWeldSpaceHeight;
        jgMoveToTcpComparison:=MergeJgWith();
        rJointGroupRound jgMoveToTcpComparison;
        IF jgMoveToTcp.Joint1=jgMoveToTcpComparison.Joint1 AND jgMoveToTcp.Joint2=jgMoveToTcpComparison.Joint2 AND jgMoveToTcp.JointG=jgMoveToTcpComparison.JointG THEN

        ELSE
            rGantry_C_Home;
            rMoveToRobotHome;
            !=====================================
            !=== Gantry Starting Postion =========
            !=====================================

            jMoveGantry:=fnCoordToJoint(fnPoseToExtax(WeldsG{1}.position));
            jMoveGantry.extax.eax_d:=nGantryAngel*(-1);
            jMoveGantry.extax.eax_c:=0;
            jMoveGantry.extax.eax_c:=Limit(0,1000,jMoveGantry.extax.eax_c);
            MoveJgJ MergeJgWith(\Gantry:=jMoveGantry),vTargetSpeed,z200;
            WaitRob\ZeroSpeed;


            jTempReadyGroup:=MergeJgWith();
            jTempReadyGroup.Joint1.robax.rax_2:=jJointStepArray{6}.robax.rax_2;
            jTempReadyGroup.Joint1.robax.rax_3:=jJointStepArray{6}.robax.rax_3;
            jTempReadyGroup.Joint1.robax.rax_4:=jJointStepArray{6}.robax.rax_4;
            jTempReadyGroup.Joint1.robax.rax_5:=jJointStepArray{6}.robax.rax_5;
            jTempReadyGroup.Joint1.robax.rax_6:=jJointStepArray{6}.robax.rax_6;

            jTempReadyGroup.Joint2.robax.rax_2:=jJointStepArray{6}.robax.rax_2;
            jTempReadyGroup.Joint2.robax.rax_3:=jJointStepArray{6}.robax.rax_3;
            jTempReadyGroup.Joint2.robax.rax_4:=jJointStepArray{6}.robax.rax_4;
            jTempReadyGroup.Joint2.robax.rax_5:=jJointStepArray{6}.robax.rax_5;
            jTempReadyGroup.Joint2.robax.rax_6:=jJointStepArray{6}.robax.rax_6;

            MoveJgJ MergeJgWith(\Rob1:=jTempReadyGroup.Joint1\Rob2:=jTempReadyGroup.Joint2),vTargetSpeed,z200;

            jTempReadyGroup.Joint1.robax.rax_1:=0;
            jTempReadyGroup.Joint2.robax.rax_1:=0;
            MoveJgJ MergeJgWith(\Rob1:=jTempReadyGroup.Joint1\Rob2:=jTempReadyGroup.Joint2),vTargetSpeed,z200;

            !!! Joint move to ready pose !!!
            jReadyGantryHeightBuffer:=CJointT();

            FOR i FROM 1 TO 10 DO
                TEST i
                CASE 1,2,3,4,5:
                    jWeldPrepareR1{i}:=CJointT(\TaskName:="T_ROB1");
                    jWeldPrepareR2{i}:=CJointT(\TaskName:="T_ROB2");
                CASE 6,7,8,9,10:
                    jWeldPrepareR1{i}:=CJointT(\TaskName:="T_ROB1");
                    jWeldPrepareR1{i}.robax.rax_1:=0;

                    jWeldPrepareR2{i}:=CJointT(\TaskName:="T_ROB2");
                    jWeldPrepareR2{i}.robax.rax_1:=0;
                    !      jWeldPrepareR2{i}.extax.eax_c:=Limit(0,1000,wobjWeldLine.uframe.trans.z-((nRobWorkSpaceHeight+120)+wobjWeldLine.oframe.trans.z+nMaxPartHeightNearArray{3}+200));
                ENDTEST
                jWeldPrepareR1{i}.robax.rax_2:=jJointStepArray{i}.robax.rax_2;
                jWeldPrepareR1{i}.robax.rax_3:=jJointStepArray{i}.robax.rax_3;
                jWeldPrepareR1{i}.robax.rax_4:=jJointStepArray{i}.robax.rax_4;
                jWeldPrepareR1{i}.robax.rax_5:=jJointStepArray{i}.robax.rax_5;
                jWeldPrepareR1{i}.robax.rax_6:=jJointStepArray{i}.robax.rax_6;

                jWeldPrepareR2{i}.robax.rax_2:=jJointStepArray{i}.robax.rax_2;
                jWeldPrepareR2{i}.robax.rax_3:=jJointStepArray{i}.robax.rax_3;
                jWeldPrepareR2{i}.robax.rax_4:=jJointStepArray{i}.robax.rax_4;
                jWeldPrepareR2{i}.robax.rax_5:=jJointStepArray{i}.robax.rax_5;
                jWeldPrepareR2{i}.robax.rax_6:=jJointStepArray{i}.robax.rax_6;
            ENDFOR

            IF (NOT jJointStepArray{1}.robax=[0,0,0,0,0,0]) MoveJgJ MergeJgWith(\Rob1:=jWeldPrepareR1{1}\Rob2:=jWeldPrepareR2{1}),vTargetSpeed,zTargetZone;
            IF (NOT jJointStepArray{2}.robax=[0,0,0,0,0,0]) MoveJgJ MergeJgWith(\Rob1:=jWeldPrepareR1{2}\Rob2:=jWeldPrepareR2{2}),vTargetSpeed,zTargetZone;
            IF (NOT jJointStepArray{3}.robax=[0,0,0,0,0,0]) MoveJgJ MergeJgWith(\Rob1:=jWeldPrepareR1{3}\Rob2:=jWeldPrepareR2{3}),vTargetSpeed,zTargetZone;
            IF (NOT jJointStepArray{4}.robax=[0,0,0,0,0,0]) MoveJgJ MergeJgWith(\Rob1:=jWeldPrepareR1{4}\Rob2:=jWeldPrepareR2{4}),vTargetSpeed,zTargetZone;
            IF (NOT jJointStepArray{5}.robax=[0,0,0,0,0,0]) MoveJgJ MergeJgWith(\Rob1:=jWeldPrepareR1{5}\Rob2:=jWeldPrepareR2{5}),vTargetSpeed,zTargetZone;

            IF (NOT jJointStepArray{6}.robax=[0,0,0,0,0,0]) MoveJgJ MergeJgWith(\Rob1:=jWeldPrepareR1{6}\Rob2:=jWeldPrepareR2{6}),vTargetSpeed,zTargetZone;
            IF (NOT jJointStepArray{7}.robax=[0,0,0,0,0,0]) MoveJgJ MergeJgWith(\Rob1:=jWeldPrepareR1{7}\Rob2:=jWeldPrepareR2{7}),vTargetSpeed,zTargetZone;
            IF (NOT jJointStepArray{8}.robax=[0,0,0,0,0,0]) MoveJgJ MergeJgWith(\Rob1:=jWeldPrepareR1{8}\Rob2:=jWeldPrepareR2{8}),vTargetSpeed,zTargetZone;
            IF (NOT jJointStepArray{9}.robax=[0,0,0,0,0,0]) MoveJgJ MergeJgWith(\Rob1:=jWeldPrepareR1{9}\Rob2:=jWeldPrepareR2{9}),vTargetSpeed,zTargetZone;
            IF (NOT jJointStepArray{10}.robax=[0,0,0,0,0,0]) MoveJgJ MergeJgWith(\Rob1:=jWeldPrepareR1{10}\Rob2:=jWeldPrepareR2{10}),vTargetSpeed,zTargetZone;
            WaitRob\inpos;
            pSearchReadyGroup:=MergePgWith();
            jSearchReadyGroup:=MergeJgWith();
        ENDIF
        jTempReadyGroup:=MergeJgWith();
        jTempGantry{1}:=fnCoordToJoint(fnPoseToExtax(WeldsG{1}.position));
        jTempReadyGroup.JointG.extax.eax_c:=jTempGantry{1}.extax.eax_c;
        jTempReadyGroup.JointG.extax.eax_d:=nGantryAngel*(-1);
        MoveJgJ MergeJgWith(\Gantry:=jTempReadyGroup.JointG),vTargetSpeed,z200;

        rMoveToTcp;
        jgMoveToTcp:=MergeJgWith();
        rJointGroupRound jgMoveToTcp;

    ENDPROC

    PROC rJointGroupRound(inout jointgroup jg)
        jg.Joint1.robax.rax_1:=Round(jg.Joint1.robax.rax_1\Dec:=0);
        jg.Joint1.robax.rax_2:=Round(jg.Joint1.robax.rax_2\Dec:=0);
        jg.Joint1.robax.rax_3:=Round(jg.Joint1.robax.rax_3\Dec:=0);
        jg.Joint1.robax.rax_4:=Round(jg.Joint1.robax.rax_4\Dec:=0);
        jg.Joint1.robax.rax_5:=Round(jg.Joint1.robax.rax_5\Dec:=0);
        jg.Joint1.robax.rax_6:=Round(jg.Joint1.robax.rax_6\Dec:=0);

        jg.Joint2.robax.rax_1:=Round(jg.Joint2.robax.rax_1\Dec:=0);
        jg.Joint2.robax.rax_2:=Round(jg.Joint2.robax.rax_2\Dec:=0);
        jg.Joint2.robax.rax_3:=Round(jg.Joint2.robax.rax_3\Dec:=0);
        jg.Joint2.robax.rax_4:=Round(jg.Joint2.robax.rax_4\Dec:=0);
        jg.Joint2.robax.rax_5:=Round(jg.Joint2.robax.rax_5\Dec:=0);
        jg.Joint2.robax.rax_6:=Round(jg.Joint2.robax.rax_6\Dec:=0);

        jg.JointG.extax.eax_a:=Round(jg.JointG.extax.eax_a\Dec:=0);
        jg.JointG.extax.eax_f:=Round(jg.JointG.extax.eax_f\Dec:=0);
        jg.JointG.extax.eax_b:=Round(jg.JointG.extax.eax_b\Dec:=0);
        jg.JointG.extax.eax_c:=Round(jg.JointG.extax.eax_c\Dec:=0);
        jg.JointG.extax.eax_d:=Round(jg.JointG.extax.eax_d\Dec:=0);
    ENDPROC

    PROC rMoveToTcp()
        VAR num nTempMmps;
        VAR jointgroup jTempReadyGroup;
        stCommand:="MoveToTcp";
        WaitUntil stReact=["MoveToTcp_Ok","MoveToTcp_Ok","MoveToTcp_Ok"];
        stCommand:="";
        WaitUntil stReact=["Ready","Ready","Ready"];
        RETURN ;
    ERROR
    ENDPROC

    PROC rDefineWobjWeldLineTcp(pos posStart,pos posEnd)
        VAR pos posWeldingLineVector;
        VAR pos posUpVector:=[0,0,1];
        VAR pos posThickVector;

        VAR num nRx;
        VAR num nRy;
        VAR num nRz;

        VAR pos posStartBuffer;
        VAR pos posEndBuffer;

        posStartBuffer:=posStart;
        posEndBuffer:=posEnd;
        posWeldingLineVector:=CalcNormalVector(posStartBuffer,posEndBuffer);
        posThickVector:=CrossProd(posUpVector,posWeldingLineVector);
        rCreateMatrix posWeldingLineVector,posThickVector,posUpVector,rotationMatrix;
        rCalcEulerAngles rotationMatrix,nRx,nRy,nRz;

        wobjWeldLine:=wobj0;
        wobjWeldLine1:=wobj0;
        wobjWeldLine2:=wobj0;

        wobjWeldLine.uframe:=WobjFloor.uframe;
        wobjWeldLine.oframe.trans:=posStart;
        wobjWeldLine.oframe.rot:=OrientZYX(nRz,nRy,nRx);
        nAngleRzStore:=nRz;
        nOffsetLengthBuffer:=0;
        nWeldLineLength_R1:=nOffsetLengthBuffer*2;
        nWeldLineLength_R2:=nOffsetLengthBuffer*2;


        IF (nAngleRzStore<-90 OR 90<=nAngleRzStore) THEN
            bRobSwap:=TRUE;
            wobjWeldLine1.uframe:=[[488,-nOffsetLengthBuffer,nRobWeldSpaceHeight],[0,0.7071067812,0.7071067812,0]];
            wobjWeldLine2.uframe:=[[488,nOffsetLengthBuffer,nRobWeldSpaceHeight],[0,0.7071067812,-0.7071067812,0]];
        ELSE
            bRobSwap:=FALSE;
            wobjWeldLine1.uframe:=[[488,nOffsetLengthBuffer,nRobWeldSpaceHeight],[0,0.7071067812,-0.7071067812,0]];
            wobjWeldLine2.uframe:=[[488,-nOffsetLengthBuffer,nRobWeldSpaceHeight],[0,0.7071067812,0.7071067812,0]];
        ENDIF

        RETURN ;
    ENDPROC

    PROC rWireCut_Select()
        IF bMoveToWireCutHome=TRUE THEN
            if nMode=1 THEN
                rWirecutShot 1;
            ELSEIF nmode=2 THEN
                rWirecutShot 2;
            ELSE
                rWirecutShot 3;
            ENDIF
        ELSE
            IF (bEnableStartEndPointCorr=TRUE) THEN
                IF nMaxPartHeightNearArray{3}>800 OR nMaxPartHeightNearArray{2}>800 THEN
                    if nMode=1 THEN
                        rWirecutMove 1;
                    ELSEIF nmode=2 THEN
                        rWirecutMove 2;
                    ELSE
                        rWirecutMove 3;
                    ENDIF
                ELSE
                    if nMode=1 THEN
                        rWirecutShot 1;
                    ELSEIF nmode=2 THEN
                        rWirecutShot 2;
                    ELSE
                        rWirecutShot 3;
                    ENDIF
                ENDIF
            ELSE
                IF nMaxPartHeightNearArray{1}>800 OR nMaxPartHeightNearArray{2}>800 THEN
                    if nMode=1 THEN
                        rWirecutMove 1;
                    ELSEIF nmode=2 THEN
                        rWirecutMove 2;
                    ELSE
                        rWirecutMove 3;
                    ENDIF
                ELSE
                    if nMode=1 THEN
                        rWirecutShot 1;
                    ELSEIF nmode=2 THEN
                        rWirecutShot 2;
                    ELSE
                        rWirecutShot 3;
                    ENDIF
                ENDIF
            ENDIF
        ENDIF

    ENDPROC

    PROC rReTurnToWireCut()
        VAR jointgroup jgTemp;

        jgTemp:=MergeJgWith();
        jgTemp.Joint1.robax:=[39.7077,23.0399,30.4536,-87.5281,29.1211,122.951];
        jgTemp.Joint2.robax:=[39.5269,22.7659,30.4413,-87.1375,29.0323,122.34];
        MoveJgJ MergeJgWith(\Rob1:=jgTemp.Joint1\Rob2:=jgTemp.Joint2),v50,fine;
        WaitRob\InPos;
        WaitRob\ZeroSpeed;

    ENDPROC

    PROC rManualOriginCheck()
        VAR jointgroup jgTemp;

        rGantry_C_Home;
        IF sdo_Rob_1_MoveHome=0 OR sdo_Rob_2_MoveHome=0 THEN
            rMoveToRobotHome;
        ENDIF
        jgTemp:=MergeJgWith();
        jgTemp.JointG.extax:=ManualOrigin_Pos.JointG.extax;
        jgTemp.JointG.extax.eax_c:=0;
        MoveJgJ MergeJgWith(\Gantry:=jgTemp.JointG),[300,300,400,25],fine;
        WaitRob\InPos;
        WaitRob\ZeroSpeed;
        MoveJgJ MergeJgWith(\Gantry:=ManualOrigin_Pos.JointG),[300,300,100,25],fine;
        WaitRob\InPos;
        WaitRob\ZeroSpeed;

    ENDPROC


ENDMODULE
